(* PLC project  *)

PROGRAM P
  VAR
    CTU_0 : CTU;
  END_VAR
  VAR  (* added by the conversion: wires and edge detectors of the diagram *)
    R_TRIG1 : R_TRIG;
  END_VAR

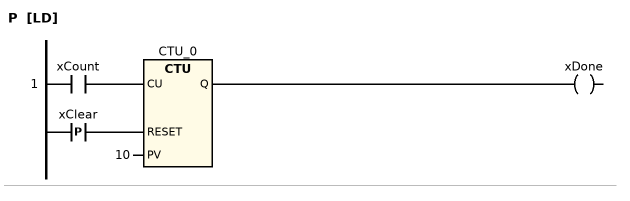
(* LD diagram, written out as Structured Text *)
R_TRIG1(CLK := xClear);
CTU_0(CU := xCount, RESET := R_TRIG1.Q, PV := 10);
xDone := CTU_0.Q;
END_PROGRAM
